(* CoDeSys 2.3 export: WATERFLOWMETER.EXP *)

(* POU PRG/WaterFlowMeter, ST *)
PROGRAM WaterFlowMeter
VAR
	WaterFlowMetr : CTU;

END_VAR
A1_DI_FlowWater;
WaterFlowMetr();
END_PROGRAM
